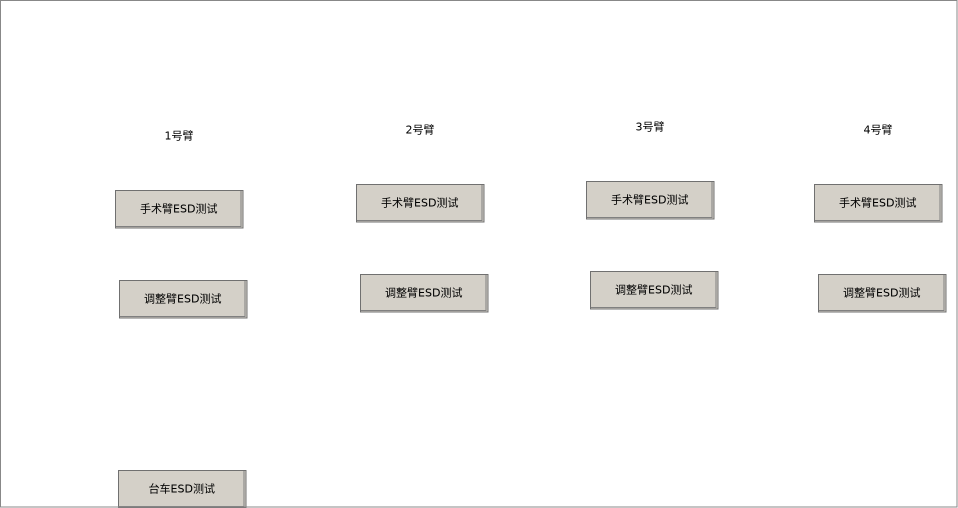
VISUALIZATION cycle_ESD  // 958x508
    Button (115,190 128x38), "手术臂ESD测试", colour toggle: g_cycleTest.m_enterESDTest[1]
        toggle g_cycleTest.m_enterESDTest[1]
    Button (119,280 128x38), "调整臂ESD测试", colour toggle: g_cycleTest.m_enterESDTestSetup[1]
        toggle g_cycleTest.m_enterESDTestSetup[1]
    Button (118,470 128x38), "台车ESD测试", colour toggle: g_cycleTest.m_carEnterESDTest
        toggle g_cycleTest.m_carEnterESDTest
    Label (99,105 160x62), "1号臂"
    Button (356,184 128x38), "手术臂ESD测试", colour toggle: g_cycleTest.m_enterESDTest[2]
        toggle g_cycleTest.m_enterESDTest[2]
    Button (360,274 128x38), "调整臂ESD测试", colour toggle: g_cycleTest.m_enterESDTestSetup[2]
        toggle g_cycleTest.m_enterESDTestSetup[2]
    Label (340,99 160x62), "2号臂"
    Button (586,181 128x38), "手术臂ESD测试", colour toggle: g_cycleTest.m_enterESDTest[3]
        toggle g_cycleTest.m_enterESDTest[3]
    Button (590,271 128x38), "调整臂ESD测试", colour toggle: g_cycleTest.m_enterESDTestSetup[3]
        toggle g_cycleTest.m_enterESDTestSetup[3]
    Label (570,96 160x62), "3号臂"
    Button (814,184 128x38), "手术臂ESD测试", colour toggle: g_cycleTest.m_enterESDTest[4]
        toggle g_cycleTest.m_enterESDTest[4]
    Button (818,274 128x38), "调整臂ESD测试", colour toggle: g_cycleTest.m_enterESDTestSetup[4]
        toggle g_cycleTest.m_enterESDTestSetup[4]
    Label (798,99 160x62), "4号臂"
END_VISUALIZATION

(* stored: Version 1.1.0.1, ProductVersion 3.1.4024.11
   Visu cycle_ESD: Id {34adcf79-bd4a-4458-9531-add87fd1bff1} *)
